(* IEC 61131-3 sources: Lasal/CPU_5344_V01/Class/BlinkLamp, 1 file *)

(* ---- BlinkLamp.st ---- *)
(*!
<Class
	Name               = "BlinkLamp"
	Revision           = "0.0"
	RealtimeTask       = "false"
	CyclicTask         = "true"
	DefCyclictime      = "100 ms"
	BackgroundTask     = "false"
	Sigmatek           = "false"
	OSInterface        = "false"
	HighPriority       = "false"
	Automatic          = "false"
	UpdateMode         = "Prescan"
	SharedCommandTable = "true"
	Objectsize         = "(284,120)">
	<Channels>
		<Server Name="ClassSvr" Visualized="false" Initialize="false" WriteProtected="true" Retentive="false"/>
		<Server Name="T_Interval" Visualized="false" Initialize="true" DefValue="500" WriteProtected="false" Retentive="false"/>
	</Channels>
</Class>
*)
BlinkLamp : CLASS
  //Servers:
	ClassSvr 	: SvrChCmd_DINT;
	T_Interval 	: SvrCh_UDINT;
  //Clients:
  //Variables:
		mBlink2 	: DINT;
		tBlink2 	: UDINT;
  //Functions:

	FUNCTION VIRTUAL GLOBAL CyWork
		VAR_INPUT
			EAX 	: UDINT;
		END_VAR
		VAR_OUTPUT
			state (EAX) 	: UDINT;
		END_VAR;
  //Tables:
	FUNCTION @STD
		VAR_OUTPUT
			ret_code	: CONFSTATES;
		END_VAR;
	FUNCTION GLOBAL TAB @CT_;
END_CLASS;

// JdK 10-2-2020: opgenomen in library, herkomst onbekend

FUNCTION VIRTUAL GLOBAL BlinkLamp::CyWork
	VAR_INPUT
		EAX 	: UDINT;
	END_VAR
	VAR_OUTPUT
		state (EAX) 	: UDINT;
	END_VAR

  if ops.tAbsolute - tBlink2 > T_Interval then
    mBlink2 := mBlink2 = 0;
    tBlink2 := ops.tAbsolute;
  end_if;

  ClassSvr := mBlink2;

	state := READY;

END_FUNCTION
